// TIA Portal V20 export
// export: Created 2025-12-01T14:57:13.5818116Z, ExportSetting None, DisplayName Totally Integrated Automation Portal, DisplayVersion V20 Update 3, DisplayName TIA Portal Openness, DisplayVersion V20 Update 3, DisplayName TIA Portal Version Control Interface, DisplayVersion V20 Update 3, DisplayName STEP 7 Professional, DisplayVersion V20 Update 3, DisplayName STEP 7 Safety, DisplayVersion V20 Update 2, DisplayName WinCC Basic/Comfort/Advanced, DisplayVersion V20 Update 3, DisplayName WinCC Professional, DisplayVersion V20 Update 3, DisplayName WinCC Unified, DisplayVersion V20 Update 3
FUNCTION "FC705_JDT02AnalisisEnviados" : Void   // FC705, LAD
TITLE = "AnalisisEnviados" - Prepara el Mensaje KA o Lista de Eventos
{ S7_Optimized_Access := 'FALSE' }
AUTHOR : TRACKING
NAME : 20160525
VERSION : 4.1
// - Inicilizar
// - Distribucion
// - Reenviar Mensaje Anterior
// - Emitir Mensaje PING - Keep Alive
// - Emitir Nueva Lista de Eventos
// stored: AutoNumber false, SetENOAutomatically false
   VAR_TEMP
      DBUltimoEmi : Word;   // Num. DB del Ultimo Mensaje Emitido
      DBEventosEmi : Word;   // Num. DB de la Lista de Eventos Generados (Emitir)
      Longitud : UDInt;
      ReturnValor : Int;
      IdentEmisor : DInt;
      IdentReceptor : DInt;
      TMPEsperaAK : UDInt;
      TMPEnvioKA : UDInt;
   END_VAR
BEGIN

NETWORK
TITLE = Inicilizar
// - Inicializar Variables de los DB's
// - Coger de la configuracion el Identificador del Emisor (12)
// - Coger de la configuracion el Identificador del Receptor (18)
// - Temporizador de Espera ACKN - Confirmacion
// - Temporizador de Emision PING - Keep Alive
// - Mirar si el enlace esta activo
// -------------------------------------------------------------------------------------------
// Si trabaja sin Agencia  2016 05 25
      SET;
      A     "Activar_JDT02";  // Mirar si se trabaja con agencia
      JC    ExisteAngencia;  // modificacion nieves el 28/03/18

// Si no hay mensaje no borrar
      L     "DB707_JDT02EventosGenerados".Mensaje[0];
      L     0;
      ==I;
      JC    Final;

      CALL  "FC898_BorrarMensaje"
      ( DB_A_RESET := "DB707_JDT02EventosGenerados"  // ¿Hay que borrarlo asi?
      );  // Damos por acabado EventosGenerados

      JU    Final;  // Se ha finalizado

ExisteAngencia:NOP   0;

// -------------------------------------------------------------------------------------------
// Inicializar Variables de los DB's

      L     "JDT2_NDB_UltimoEmi";  // Cogemos el DB de UltimoEnviado
      T     #DBUltimoEmi;
      L     "JDT2_NDB_EventosEmi";  // Cogemos el DB de EventosGenerados
      T     #DBEventosEmi;


// --------------------------------------------------------------------------------------------
// Coger de la configuracion el Idendificador del emisor

      L     "JDT2_IdentEmisor";
      T     #IdentEmisor;

// --------------------------------------------------------------------------------------------
// Coger de la configuracion el Idendificador del receptor

      L     "JDT2_IdentReceptor";
      T     #IdentReceptor;

// -------------------------------------------------------------------------------------------
// Mirar si el enlace esta activo

      AN    "DB701_JDT02StatusCOM".EnlaceCP_OK;
      JC    Final;  // El EnlaceCP esta NOK, no hacer nada

// -------------------------------------------------------------------------------------------
// Temporizador de Espera PING - Confirmacion del Mensaje enviado, para el reenvio de Mensaje

      L     "JDT2_TMPEsperaAK";
      T     #TMPEsperaAK;
      CALL  "FC899_TMP"
      ( Temporizar     := "DB701_JDT02StatusCOM".EsperandoAK,
        Valor_Tiempo   := #TMPEsperaAK,  // Tiempo de 10 Segundos
        Base_tiempo_ms := 1000,
        Tiempo_OK      := "DB701_JDT02StatusCOM".TMPEsperaAK_OK,
        Valor_Actual   := "DB701_JDT02StatusCOM".TMPEsperaAK
      );

// -------------------------------------------------------------------------------------------
// Temporizador de Emision PING - Keep Alive (Si no hay actividad)

      L     "JDT2_TMPEnvioKA";
      T     #TMPEnvioKA;
      CALL  "FC899_TMP"
      ( Temporizar     := "DB701_JDT02StatusCOM".SinActividad,
        Valor_Tiempo   := #TMPEnvioKA,  // Tiempo de 1 Minuto
        Base_tiempo_ms := 1000,
        Tiempo_OK      := "DB701_JDT02StatusCOM".TMPEnvioKA_OK,
        Valor_Actual   := "DB701_JDT02StatusCOM".TMPEnvioKA
      );


NETWORK
TITLE = Distribucion
// - Miro si el mensaje anterior esta enviado correctamente
// - Mirar si es mensaje de lista de eventos, para tener que reenvialo
// - Miramos si Hay que Emitir Lista de Eventos
// - Miramos si ha pasado el tiempo para emitir el mensaje PING - Keep Alive
// -------------------------------------------------------------------------------------------
// 1º Paso - Miro si el mensaje anterior esta enviado correctamente
      L     0;
      LAR1;
      OPN   DB [#DBUltimoEmi];
      L     DBB [AR1, P#0.0];
      L     0;
      ==I;  // Esta Tratado el mensaje anterior
      JC    SiguienteMensaje;  // Ir a tratar el siguiente

// -------------------------------------------------------------------------------------------
// 2º Paso - No esta libre. Hay que ver si el Anterior Mensaje es de Lista de eventos
//           Para ver si hay que reenviar el Mensaje

      OPN   DB [#DBUltimoEmi];
      L     DBB [AR1, P#0.0];
      L     'N';  // Si tiene 'N' es un Mensaje de Lista de Eventos
      ==I;
      JC    EmisionEvento_ReEnviar;  // Ir Emitir Reenvio del Evento si es necesario

      SET;  // No se ha emitido todavia
      R     "DB701_JDT02StatusCOM".EsperandoAK;
      JU    Final;  // No hay nada todavia

// -------------------------------------------------------------------------------------------
// 3º Paso - Esta libre. Miramos si Hay que Emitir Lista de Eventos

SiguienteMensaje:L     0;  // Mirar si hay Lista de Eventos a Emitir
      LAR1;
      OPN   DB [#DBEventosEmi];
      L     DBB [AR1, P#0.0];
      L     '{';
      ==I;
      JC    EmisionEvento_ListaDeEventos;  // Ir a Emitir Nueva Lista de Eventos

// -------------------------------------------------------------------------------------------
// 4º Paso - No hay actividad. Miramos si ha pasado el tiempo para emitir el mensaje KA
      SET;
      S     "DB701_JDT02StatusCOM".SinActividad;

      A     "DB701_JDT02StatusCOM".TMPEnvioKA_OK;
      JC    EmisionEvento_KeepAlive;  // Ir a Emitir el Mensaje KA

      JU    Final;  // No va hacerse nada por ahora




NETWORK
TITLE = Reenvio del Mensaje Anterior
// - Mirar si ha pasaso el Tiempo de Espera del Mensaje ACKN - Confirmacion
// - Reenviar el Mensaje Anterior
EmisionEvento_ReEnviar:NOP   0;

// -------------------------------------------------------------------------------------------
// 1º Paso - Mirar si ha pasado el tiempo de Espera del Mensaje AK - Confirmacion

      SET;
      S     "DB701_JDT02StatusCOM".EsperandoAK;

      AN    "DB701_JDT02StatusCOM".TMPEsperaAK_OK;
      JC    Final;

// -------------------------------------------------------------------------------------------
// Reeenviar el mensaje anterior
// Solo Cambiar el primer digito 'N' -> 0x02


//Nieves 26/05/25 Control de los reintentos

// evaluamos si ya hemos intentado emitir el mensaje 3 veces
      SET;
      L     "Reintentos_JDT2";
      L     3;
      <=I;
      JC    reintenta;

// si ya hemos llegado a 3 reintentos, forzamos la desconexión

      L     1;
      T     "Reintentos_JDT2";
      SET;
      S     "DB701_JDT02StatusCOM".EmiJdT_Reset;
      JU    Final;  // Se ha finalizado

reintenta:NOP   0;
      L     "Reintentos_JDT2";
      L     1;
      +I;
      T     "Reintentos_JDT2";



// fin control reintentos


      SET;  // Voy ha Reenviar el Mensaje
      R     "DB701_JDT02StatusCOM".EsperandoAK;  // Con esto reseto el timer

      L     0;
      LAR1;
      OPN   DB [#DBUltimoEmi];  // Cambio el inicio del Mensaje
      L     2;
      T     DBB [AR1, P#0.0];

      JU    Final;  // Se ha finalizado


NETWORK
TITLE = Emitir PING - Keep Alive
// - Resetear variables
// - Formateo del Mensaje PING - Keep Alive
EmisionEvento_KeepAlive:NOP   0;
      O;
// -------------------------------------------------------------------------------------------
// 1º Paso - Resetear variables

      SET;  // Si hay Actividad
      R     "DB701_JDT02StatusCOM".SinActividad;  // Con esto reseto el timer

// -------------------------------------------------------------------------------------------
// 2º Paso - Formateo en Mensaje KA - Con el ultimo secuencial

// Numero Secuencial - Con el ultimo secuencial

      CALL  "FC891_EtiqDInt_EtiqChar"
      ( DB_String   := "JDT2_NDB_UltimoEmi",  // DB UltimoEmision
        Long_String := 4,
        Offset_Ini  := 4,
        Valor       := "DB701_JDT02StatusCOM".ID_UltimoEnviado
      );  // Rellenar el ID del Mensaje

      L     0;  // Puntero DB UltimoEmision
      LAR1;
      OPN   DB [#DBUltimoEmi];

      L     2;  // Primer Byte 0x02 - Para que sea enviada
      T     DBB [AR1, P#0.0];
      L     ';';  // Separador
      T     DBB [AR1, P#5.0];

      L     #IdentEmisor;  // Rellenar el Campo Emisor
      T     DBD [AR1, P#6.0];

      L     ';';  // Separador
      T     DBB [AR1, P#10.0];

      L     #IdentReceptor;  // Rellenar el Campo Receptor
      T     DBD [AR1, P#11.0];

      L     ';';  // Separador
      T     DBB [AR1, P#15.0];

      L     '0';  // Campo Tamaño del Mensaje
      T     DBB [AR1, P#16.0];  // En dos partes '0' y '0031'
      L     '0031';
      T     DBD [AR1, P#17.0];

      L     ';';  // Separador
      T     DBB [AR1, P#21.0];

// Evento  a escrribir- ({KA})

      L     '({';  // Empieza Evento
      T     DBW [AR1, P#22.0];
      L     'PING';  // Evento AK
      T     DBD [AR1, P#24.0];
      L     '})';  // Final del Evento
      T     DBW [AR1, P#28.0];

      L     3;  // Final del Mensaje 0x03
      T     DBB [AR1, P#30.0];

      JU    Final;  // Se ha finalizado


NETWORK
TITLE = Emitir Nueva Lista de Eventos
// - Obtener nuevo numero secuencial
// - Formateo de la Cabecera del Mensaje
// - Formateo del Cuerpo del Mensaje - Lista de Eventos
// - Formateo el final del Mensaje
EmisionEvento_ListaDeEventos:NOP   0;

// -------------------------------------------------------------------------------------------
// 1º Paso - Obtener nuevo numero secuencial

      L     "DB701_JDT02StatusCOM".ID_UltimoEnviado;
      L     1;  // Se Suma +1
      +D;
      T     "DB701_JDT02StatusCOM".ID_UltimoEnviado;  // Guardo el Nuevo ID

      L     "DB701_JDT02StatusCOM".ID_UltimoEnviado;
      L     9999;  // Ha pasado el Limite
      <=I;
      JC    _050;

      L     1;  // Empieza de nuevo
      T     "DB701_JDT02StatusCOM".ID_UltimoEnviado;  // Guardo el Nuevo ID

_050: L     "DB701_JDT02StatusCOM".ID_UltimoEnviado;
      T     #ReturnValor;  // Valor del ID del Mensaje

// -------------------------------------------------------------------------------------------
// 2º Paso -  Formateo de la Cabecera del Mensaje
// Nota: Faltara el tamaño del mensaje que se hara al final

      CALL  "FC891_EtiqDInt_EtiqChar"
      ( DB_String   := "JDT2_NDB_UltimoEmi",  // DB UltimoEmision
        Long_String := 4,
        Offset_Ini  := 4,
        Valor       := "DB701_JDT02StatusCOM".ID_UltimoEnviado
      );  // Rellenar el ID del Mensaje

      L     0;  // Puntero DB UltimoEmision
      LAR1;

      OPN   DB [#DBUltimoEmi];
      L     2;  // Primer Byte 0x02 - Para que sea enviada
      T     DBB [AR1, P#0.0];
      L     ';';  // Separador
      T     DBB [AR1, P#5.0];


      L     #IdentEmisor;  // Rellenar el Campo Emisor
      T     DBD [AR1, P#6.0];

      L     ';';  // Separador
      T     DBB [AR1, P#10.0];

      L     #IdentReceptor;  // Rellenar el Campo Receptor
      T     DBD [AR1, P#11.0];

      L     ';';  // Separador
      T     DBB [AR1, P#15.0];

// Falta el tamaño que se rellenara con el final

      L     ';';  // Separador
      T     DBB [AR1, P#21.0];

      L     '(';  // Inicio de la Lista de Eventos
      T     DBB [AR1, P#22.0];

// -------------------------------------------------------------------------------------------
// 3º Paso -  Formateo del Cuerpo del Mensaje - Lista de Eventos

      +AR1  P#23.0;  // AR1 = PunteroDestino
      L     0;  // AR2 = PunteroOrigen
      LAR2;

_051: OPN   DB [#DBEventosEmi];  // Transferir los datos
      L     DBB [AR2, P#0.0];  // De Origen
      OPN   DB [#DBUltimoEmi];
      T     DBB [AR1, P#0.0];  // A Destino

      L     0;  // Si es 0 - Ha llegado al final de la lista de Eventos
      ==I;
      JC    _052;  // Si Ha llegado al final

      +AR1  P#1.0;  // Se incrementa los punteros
      +AR2  P#1.0;
      JU    _051;

// -------------------------------------------------------------------------------------------
// 4º Paso -  Formateo del Final del Mensaje

_052: OPN   DB [#DBUltimoEmi];
      L     ')';  // Final de la Lista de Eventos
      T     DBB [AR1, P#0.0];

      L     3;  // Ultimo Byte - 0x03
      T     DBB [AR1, P#1.0];

// -------------------------------------------------------------------------------------------
// 5º Paso - Poner el tamaño del Mensaje

      TAR1;  // Calculo el Tamaño del Mensaje
      SRD   3;
      L     2;  // Añadir los dos ultimos digitos
      +D;
      T     #Longitud;

      CALL  "FC891_EtiqDInt_EtiqChar"
      ( DB_String   := "JDT2_NDB_UltimoEmi",  // DB UltimoEmision
        Long_String := 5,
        Offset_Ini  := 20,
        Valor       := #Longitud
      );  // Rellenar el Campo Tamaño del mensaje

// -------------------------------------------------------------------------------------------
// 6º Paso - Limpio las variables

      SET;
      S     "DB701_JDT02StatusCOM".EsperandoAK;

      CALL  "FC898_BorrarMensaje"
      ( DB_A_RESET := "DB707_JDT02EventosGenerados"  // ¿Hay que borrarlo asi?
      );  // Damos por acabado EventosGenerados

      JU    Final;  // Se ha finalizado


NETWORK
TITLE = Finalizar
// Se acabo la funcion
Final:NOP   0;

END_FUNCTION
